# EPICS alarm handler configuration: alh_files/mgnt_li21L2.alhConfig
GROUP NULL MGNT:LI21L2:1
   $COMMAND edm -x -eolc -noedit mgnt_li21_main.edl

$ALIAS LI21L2
$GUIDANCE
li21L2 Magnets
   Group Name: MGNT:LI21L2:1
   Summary PV:  MGNT:LI21L2:1:STATSUMY
$END

   INCLUDE MGNT:LI21L2:1 ./mgnt_li21L2_lgps.alhConfig
   INCLUDE MGNT:LI21L2:1 ./mgnt_li21L2_quad.alhConfig
   INCLUDE MGNT:LI21L2:1 ./mgnt_li21L2_xcor.alhConfig
   INCLUDE MGNT:LI21L2:1 ./mgnt_li21L2_ycor.alhConfig
